INTERFACE IStation

PROPERTY Position : REFERENCE TO FB_Position
GET
END_GET
SET
END_SET
END_PROPERTY

PROPERTY Process : REFERENCE TO FB_AUT_ABSTRACT
GET
END_GET
SET
END_SET
END_PROPERTY

END_INTERFACE

(* stored: Version 1.1.0.1, ProductVersion 3.1.4024.12
   Itf IStation: Id {1b1cfc52-067c-4cca-bb54-8b1837d35537}
   Property Position: Id {d5fdfcdc-e558-4dc2-a053-aa38137ac309}
   Get Get: Id {eb1908f7-bb26-4e96-95d4-32f8a81443af}
   Set Set: Id {41e537a6-6b8d-4feb-a977-c6dfcf7a7de7}
   Property Process: Id {130396d9-b675-443f-bd6b-1fece5b4a368}
   Get Get: Id {95998982-ad2e-4b3f-88fa-5bac9383cce1}
   Set Set: Id {64385389-36af-4228-a699-aa8f1352a8c4} *)
